// TwinCAT 3 PLC project SimulationProject
// ProgramVersion: 3.1.4024.0
// libraries:
//   Tc2_Standard, * (Beckhoff Automation GmbH)
//   Tc2_System, * (Beckhoff Automation GmbH)
//   Tc3_Module, * (Beckhoff Automation GmbH)
//   VisuSymbols,3.5.10.0,System
// project tree:
//   DUTs/ cylinder2IO.TcDUT, position_status.TcDUT, _2_position.TcDUT
//   / GlobalTextList.TcGTLO, PlcTask.TcTTO, Visualization Manager.TcVMO (not stored)
//   POUs/ Cylinder.TcPOU, SimulationMAIN.TcPOU
//   VISUs/ Visualization.TcVIS
// (motion and I/O tree: see PLC project developmentproject)
// real-time tasks:
//   TASK PlcTask: cycle T#10ms, priority 20, ADS port 350
//   TASK PlcTask1: cycle T#5ms, priority 21, ADS port 351
// variable links:
//   SimulationProject/SimulationProject Instance <-> Device 1 (EtherCAT Simulation)/Term 2 (EL1012)
//     PlcTask Outputs/SimulationMAIN.io._pull_sensor <-> Channel 2/Input
//     PlcTask Outputs/SimulationMAIN.io._push_sensor <-> Channel 1/Input
//   SimulationProject/SimulationProject Instance <-> Device 1 (EtherCAT Simulation)/Term 4 (EL2004)
//     PlcTask Inputs/SimulationMAIN.io._pull_output <-> Channel 2/Output
//     PlcTask Inputs/SimulationMAIN.io._push_output <-> Channel 1/Output

CONFIGURATION SimulationProject
    RESOURCE PLC ON TwinCAT3
        TASK PlcTask(INTERVAL := T#5ms, PRIORITY := 21);
        PROGRAM SimulationMAIN WITH PlcTask : SimulationMAIN;
    END_RESOURCE
END_CONFIGURATION

// ---- DUTs/cylinder2IO.TcDUT
TYPE cylinder2IO :
STRUCT
	_pull_sensor	AT%Q*	:BOOL;
	_push_sensor	AT%Q*	:BOOL;
	_pull_output 	AT%I*	:BOOL;
	_push_output 	AT%I*	:BOOL;
END_STRUCT
END_TYPE

// ---- DUTs/position_status.TcDUT
{attribute 'qualified_only'}
{attribute 'strict'}
TYPE position_status :
(
	unknown := 0,
	inposition,
	moving
);
END_TYPE

// ---- DUTs/_2_position.TcDUT
{attribute 'qualified_only'}
{attribute 'strict'}
TYPE _2_position :
(
	position_1 := 0,
	position_1_2,
	position_2
);
END_TYPE

// ---- POUs/SimulationMAIN.TcPOU
PROGRAM SimulationMAIN
VAR
	cylinder_stub:	Cylinder;
	io: cylinder2IO;
	push_stroke_time: REAL := 1.8;
	pull_stroke_time: REAL := 1.5;
	chattering_time: REAL := 0.5;
END_VAR

cylinder_stub.push_time := REAL_TO_TIME(push_stroke_time * 1000);
cylinder_stub.pull_time := REAL_TO_TIME(pull_stroke_time * 1000);
cylinder_stub.chattering_time := REAL_TO_TIME(chattering_time * 1000);

cylinder_stub(io:= io);

END_PROGRAM

// ---- POUs/Cylinder.TcPOU
FUNCTION_BLOCK Cylinder
VAR_INPUT
	push_time: TIME := T#3S;
	pull_time: TIME := T#1S;
	push_release_time: TIME := T#150MS;
	pull_release_time: TIME := T#150MS;
	chattering_push: BOOL := TRUE;
	chattering_pull: BOOL := TRUE;
	chattering_time: TIME := T#2S;
	chattering_hl_time: TIME := T#50MS;
END_VAR
VAR_OUTPUT
END_VAR
VAR
	push_timer: Tc2_Standard.TON;
	pull_timer: Tc2_Standard.TON;
	chattering_gen: Tc2_Standard.TP;
	_chattering_gen: Tc2_Standard.TP;
	chattering_timer: Tc2_Standard.TON;
	
END_VAR

VAR_IN_OUT
	io: cylinder2IO;
END_VAR


push_timer(IN:=(io._push_output AND NOT io._pull_output), PT:= push_time);
pull_timer(IN:=(io._pull_output AND NOT io._push_output), PT:= pull_time);

IF push_timer.Q THEN
	IF chattering_push THEN
		chattering_timer(IN:=TRUE, PT:=chattering_time);
		IF chattering_timer.Q THEN
			io._push_sensor := TRUE;
		ELSE
			chattering_gen(IN:=NOT _chattering_gen.Q, PT:=chattering_hl_time);
			_chattering_gen(IN:=NOT chattering_gen.Q, PT:=chattering_hl_time);
			io._push_sensor := chattering_gen.Q;
		END_IF
	ELSE
		io._push_sensor := TRUE;
	END_IF	 
END_IF


IF pull_timer.Q THEN
	IF chattering_pull THEN
		chattering_timer(IN:=TRUE, PT:=chattering_time);
		IF chattering_timer.Q THEN
			io._pull_sensor := TRUE;
		ELSE
			chattering_gen(IN:=NOT _chattering_gen.Q, PT:=chattering_hl_time);
			_chattering_gen(IN:=NOT chattering_gen.Q, PT:=chattering_hl_time);
			io._pull_sensor := chattering_gen.Q;
		END_IF
	ELSE
		io._pull_sensor := TRUE;
	END_IF	 
END_IF

IF 	NOT push_timer.Q AND NOT pull_timer.Q THEN
	chattering_gen(IN:=FALSE);
	chattering_timer(IN:=FALSE);
END_IF


IF pull_timer.ET > push_release_time THEN
	io._push_sensor := FALSE;
END_IF

IF push_timer.ET > pull_release_time THEN
	io._pull_sensor := FALSE;	
END_IF

END_FUNCTION_BLOCK

// ---- GlobalTextList.TcGTLO
TEXTLIST GlobalTextList
  544 = '%0.1f'
  710 = 'Chattering high time'
  128 = 'Chattering term'
  443 = 'Chattering time'
  997 = 'ms'
  198 = 'Over time'
  781 = 'Pull chattering'
  138 = 'Pull relase time'
  878 = 'Pull stabilization'
  192 = 'Pull stroke time'
  333 = 'Push chattering'
  801 = 'Push relase time'
  548 = 'Push stroke time'
  545 = 's'
END_TEXTLIST

// ---- VISUs/Visualization.TcVIS
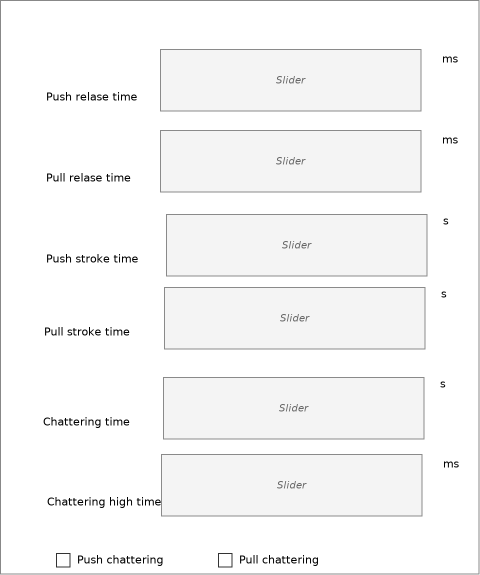
VISUALIZATION Visualization  // 480x575
    Label (43,82 150x30), "Push relase time"
    Slider (160,49 261x62), variable: SimulationMAIN.cylinder_stub.push_release_time, scale 0..1000
    Label (439,44 40x30), "ms"
    Label (43,163 150x30), "Pull relase time"
    Slider (160,130 261x62), variable: SimulationMAIN.cylinder_stub.pull_release_time, scale 0..1000
    Label (439,125 40x30), "ms"
    Slider (166,214 261x62), variable: SimulationMAIN.push_stroke_time, scale 0..10
    Label (43,244 150x30), "Push stroke time"
    Label (440,206 40x30), "s"
    Slider (164,287 261x62), variable: SimulationMAIN.pull_stroke_time, scale 0..10
    Label (41,317 150x30), "Pull stroke time"
    Label (438,279 40x30), "s"
    Slider (163,377 261x62), variable: SimulationMAIN.chattering_time, scale 0..5
    Label (40,407 150x30), "Chattering time"
    Label (437,369 40x30), "s"
    Label (44,487 150x30), "Chattering high time"
    Slider (161,454 261x62), variable: SimulationMAIN.cylinder_stub.chattering_hl_time, scale 0..100
    Label (440,449 40x30), "ms"
    Checkbox (54,545 150x30), "Push chattering", variable: SimulationMAIN.cylinder_stub.chattering_push
    Checkbox (216,545 150x30), "Pull chattering", variable: SimulationMAIN.cylinder_stub.chattering_pull
END_VISUALIZATION
